Fanuc KAREL source: kt00204.KL

-- PROVISIONAL review KL for V940-1; original PC SHA256 50d278b7af3618ff6f6bd23f8c3bce4d5ded7d027daeb2f5f165ade455bebb3f
-- Incomplete behavior may be omitted. Consult companion uncertainty JSON. Do not deploy.
PROGRAM KT00204
%NOLOCKGROUP
VAR
  I1 : INTEGER
  I2 : INTEGER
  OUT : INTEGER
BEGIN
  -- V9_ZERO_TABLE_METADATA_HINT layout=0001; no indexed target words; source/name/runtime held
  -- UNRESOLVED_PC offsets 5-16; opcodes 2E,23
  -- UNRESOLVED_PC offsets 21-32; opcodes 2E,23
  -- UNRESOLVED_PC offsets 37-48; opcodes 2E,23
  -- UNRESOLVED_PC offsets 53-64; opcodes 2E,23
  -- UNRESOLVED_PC offsets 69-88; opcodes 21,21,46,23
  -- UNRESOLVED_PC offsets 93-97; opcodes 7F
END KT00204
